FUNCTION_BLOCK FB_ResetAll
VAR_INPUT
	execute: BOOL;
END_VAR
VAR_OUTPUT
	done: BOOL;
	busy: BOOL;
	error: BOOL;
END_VAR
VAR
	fbreset: ARRAY[1..axcnt] OF MC_Reset;
	fbgrpreset: ARRAY[1..grpcnt] OF MC_Reset;
	i: UINT;
END_VAR


done := TRUE;
busy := FALSE;
error := FALSE;

FOR i:=1 TO axcnt DO
	fbreset[i](Axis:=ax[i], Execute := execute);

	IF (NOT fbreset[i].done) THEN
		done := FALSE;
	END_IF
	IF (fbreset[i].busy) THEN
		busy := TRUE;
	END_IF
	IF (fbreset[i].Error) THEN
		error := TRUE;
	END_IF
END_FOR
FOR i:=1 TO grpcnt DO
	fbgrpreset[i](Axis:=grp[i], Execute := execute);

	IF (NOT fbgrpreset[i].done) THEN
		done := FALSE;
	END_IF
	IF (fbgrpreset[i].busy) THEN
		busy := TRUE;
	END_IF
	IF (fbgrpreset[i].Error) THEN
		error := TRUE;
	END_IF
END_FOR

END_FUNCTION_BLOCK

(* stored: Version 1.1.0.1, ProductVersion 3.1.0.25
   POU FB_ResetAll: Id {bab6a601-8b9f-40df-b6fb-5e9e0e0bbb96} *)
